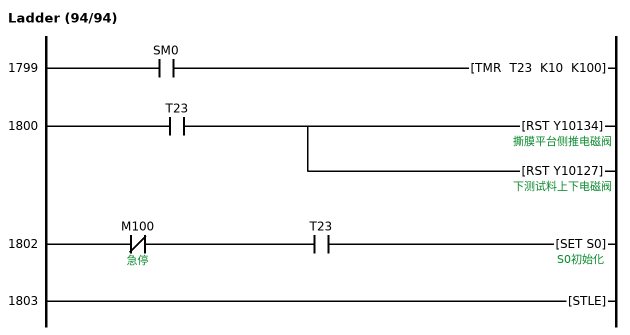
[picture p96: Ladder rows 1799-1803]
LD     SM0
TMR    T23 K10 K100
LD     T23
RST    Y10134	; 撕膜平台侧推电磁阀
RST    Y10127	; 下测试料上下电磁阀
LDI    M100	; 急停
AND    T23
SET    S0	; S0初始化
STLE

COMMENTS (devices not used above)
X10	下料有无漫反射
X13	吸料盘上下气杆置位传感器
X23	矫正负压信号2
X26	上测试料上下气缸SET传感器
X30	矫正气缸SET传感器
X32	矫正负压信号1
X37	下测试料翻转气缸SET传感器
X41	撕膜平台吸左产品膜负压信号1
X10013	撕膜平台吸右产品膜负压信号2
X10034	排料完成【自机械手】
X10036	穴1样本取料
X10037	穴2样本取料
X10300	上测试轴取料光纤信号1
X10302	上测试轴取料光纤信号2
X10304	前测试轴取料光纤信号1
X10306	前测试轴取料光纤信号2
X10310	后测试轴取料光纤信号1
X10312	后测试轴取料光纤信号2
X10314	穴1样本PASS
X10315	穴1样本FAIL
X10316	穴2样本PASS
X10317	穴2样本FAIL
X10412	进入样本模式
Y10103	上盘步进轴方向-9
Y10106	下盘步进轴方向-10
Y10204	吸废膜真空吸电磁阀1
Y10207	吸废膜真空吸电磁阀2
Y10225	照明灯控制输出
Y10233	上料位反向信号 【至机械手】
Y10236	机械手可以取矫正盘【至机械手】
Y10403	上料机尾料信号
Y10404	样本取料完成信号
Y10406	联机复位信号
Y10407	上料机报警信号
Y10412	允许灵敏度开始测试信号（灵敏测试机）
M20101	SCR-Running【机械手-运行】
M20103	SCR-Error【机械手-错误】
M20104	SCR-Estop【机械手-停止】
M20105	SCR-SafeguardOn【机械手-安全门】
M20106	SCR-SError【机械手-严重错误】
M20107	SCR-Warning【机械手-警告】
M20110	放料完成
S99	S99急停处理
D411	s
HD203	良品数
HD2009	上测试料上下气缸报警次数
HD2010	前上下测料上下气缸报警次数
HD10000	下料横移搬轴运行频率
HD10002	上测试料轴运行频率
HD10004	下测试料轴运行频率
HD10006	撕膜横移轴运行频率
HD10008	撕膜上下轴运行频率
HD10010	横移测料轴运行频率
HD10012	上下测料轴运行频率
HD10014	下料上下搬轴运行频率
HD10016	上盘步进轴运行频率
HD10018	下盘步进轴运行频率